# EPICS substitutions: ucmApp/Db/undulator/undulatorRTD.substitutions
file undulatorRTD.template{
  pattern { RTD, PORTNUM }
          {  01, 16      }
          {  02, 17      }
          {  03, 18      }
          {  04, 19      }
          {  05, 20      }
          {  06, 21      }
          {  07, 22      }
          {  08, 23      }
          {  09, 24      }
          {  10, 25      }
          {  11, 26      }
          {  12, 27      }
}
